FUNCTION_BLOCK T_SENSOR (* Temperature sensor *)
  (* Standard: 61499-2 *)
  (* Version 1.0, 2018-12-07, badger, AUT SERL EMSOFT, Original version *)
  (* Compiler header: #include "diags.h" *)
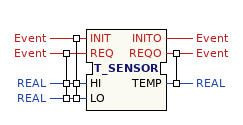
  EVENT_INPUT
    INIT WITH HI, LO; (* Initialization Request *)
    REQ WITH HI, LO; (* Normal Execution Request *)
  END_EVENT
  EVENT_OUTPUT
    INITO; (* Initialization Confirm *)
    REQO WITH TEMP; (* Signals that a new temperature reading is available. *)
  END_EVENT
  VAR_INPUT
    HI : REAL := 100; (* Maximum (highest) temperature the system will detect *)
    LO : REAL := 20; (* Minimum lowest temperature the system will detect *)
  END_VAR
  VAR_OUTPUT
    TEMP : REAL; (* Current probe temperature in F *)
  END_VAR
  VAR
    temperatureDirection : INT := 1; (* Specifies if the temperature is rising or falling. *)
  END_VAR
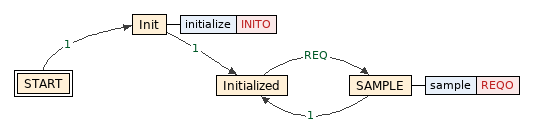
  EC_STATES
    START; (* Initial State *)
    Init : initialize -> INITO; (* Initialization *)
    SAMPLE : sample -> REQO; (* Normal execution *)
    Initialized;
  END_STATES
  EC_TRANSITIONS
    START TO Init := 1;
    Initialized TO SAMPLE := REQ;
    SAMPLE TO Initialized := 1;
    Init TO Initialized := 1;
  END_TRANSITIONS
  ALGORITHM initialize IN AnyText: (* Initialization algorithm *)
std::cout << "initialize\n";

srand(  (unsigned int)   time(NULL)   );

temperatureDirection() = 1;
srand(  (unsigned int)   TForteInt8(time(NULL))   );

if  (HI() > 0) {
	TEMP() = HI() / 2;
} else {
    if  (LO() > 0) {
			TEMP() = LO();
	 } else {
        	TEMP() = 0;
 	}
}
  END_ALGORITHM
  ALGORITHM sample IN AnyText: (* Sample the probe *)
float tempDifference = 0;

std::cout << "sample\n";

tempDifference = (static_cast<TForteFloat>(rand())/static_cast<TForteFloat>(RAND_MAX) ) * 10;
std::cout << "temperature difference =" << std::to_string(tempDifference) << "\n";

tempDifference = tempDifference * temperatureDirection();
temperatureDirection() =  - temperatureDirection();

TEMP() = TEMP() + tempDifference;
if (TEMP() > HI() ) {
	TEMP() = HI() - tempDifference;
    temperatureDirection() = -1;
} else if (TEMP() < LO() ) {
	TEMP() = LO();
    temperatureDirection() = 1;
}
  END_ALGORITHM
END_FUNCTION_BLOCK
